// TIA Portal V20 export
TYPE "typeDataFlinkUsed"
// stored: Access Published, IsFailsafeCompliant true, Namespace Safety
   STRUCT
      Cellinterlocks : "Safety.s_zc_CellInterlocks";
      Normalinterlocks : "Safety.s_zc_NormalInterlocks";
   END_STRUCT;
END_TYPE
